// TIA Portal V20 export
FUNCTION "CollectAlarms" : Void   // FC71, LAD
TITLE = U1Em7_SepaPnp
// stored: Namespace Unit1.Em7, SetENOAutomatically false
   VAR_INPUT
      resetAlarms : Bool;
      disableAlarms : Bool;
   END_VAR
   VAR_OUTPUT
      commandsToUnit : "LUC_typeStateCommands";   // Feedback to the unit
   END_VAR
   VAR CONSTANT
      DelayTime : Time := T#300ms;
      NoDelayTime : Time;
   END_VAR
BEGIN

REGION Network 1: Reset Alarms
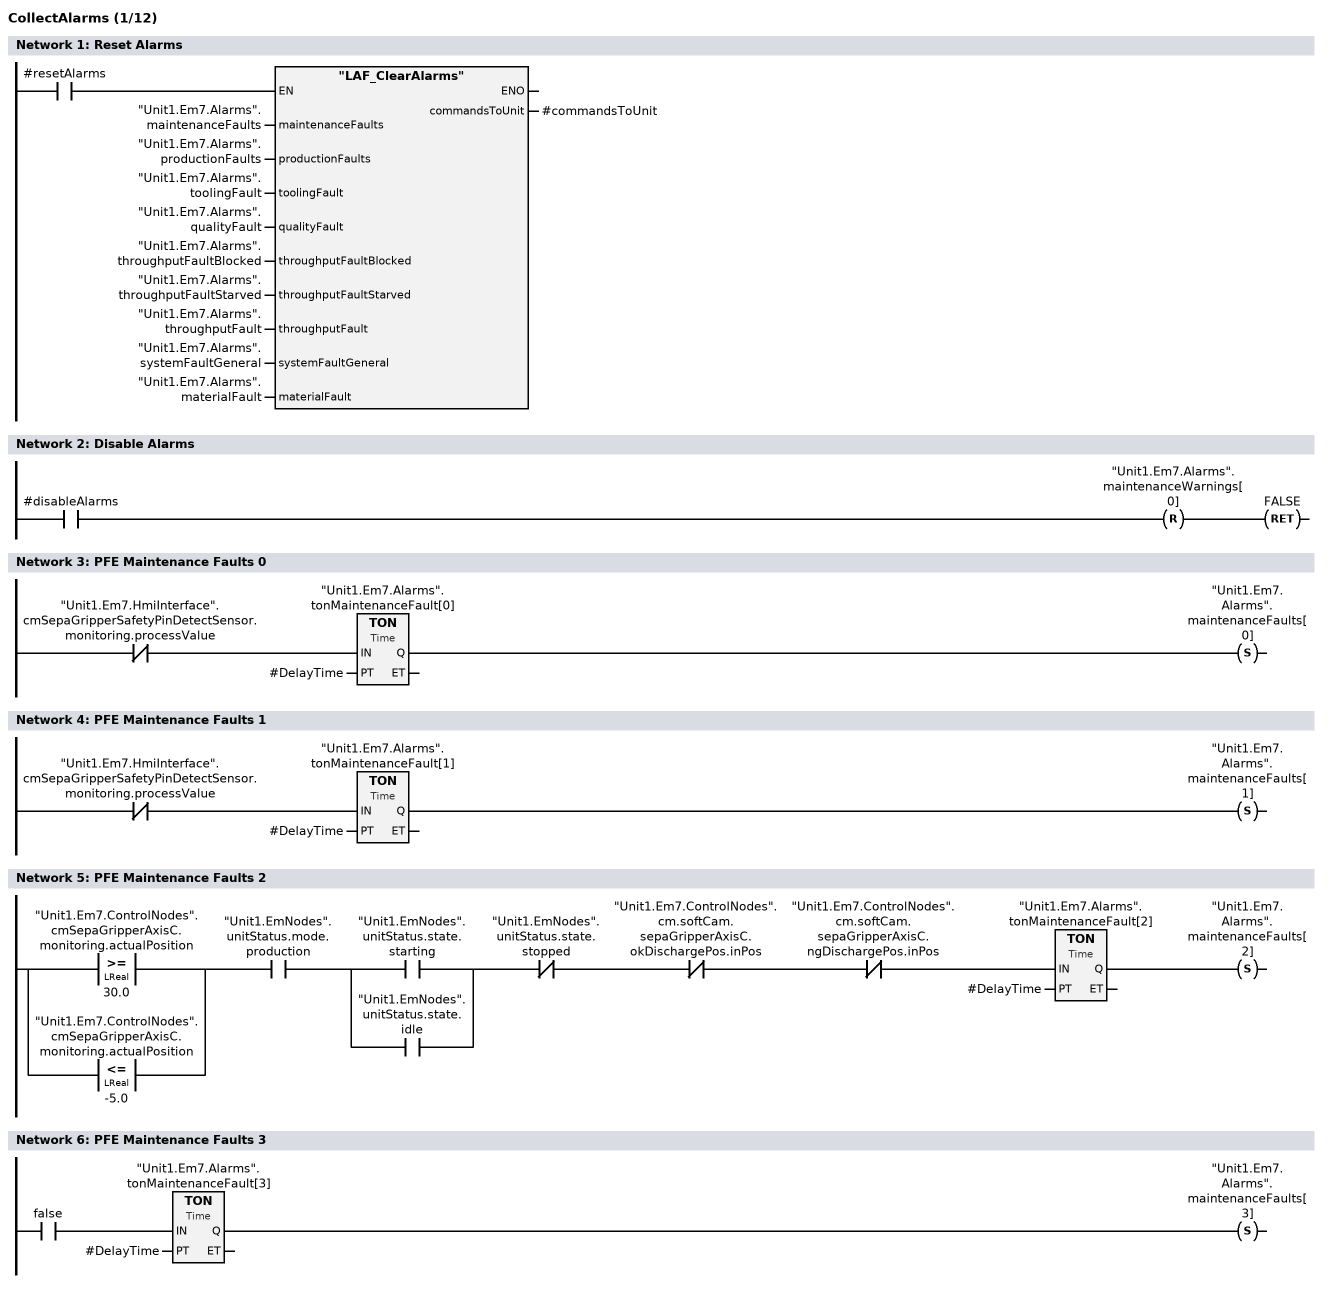
   RUNG wire#powerrail
      Contact( #resetAlarms )
      "LAF_ClearAlarms"(maintenanceFaults := "Unit1.Em7.Alarms".maintenanceFaults, productionFaults := "Unit1.Em7.Alarms".productionFaults, toolingFault := "Unit1.Em7.Alarms".toolingFault, qualityFault := "Unit1.Em7.Alarms".qualityFault, throughputFaultBlocked := "Unit1.Em7.Alarms".throughputFaultBlocked, throughputFaultStarved := "Unit1.Em7.Alarms".throughputFaultStarved, throughputFault := "Unit1.Em7.Alarms".throughputFault, systemFaultGeneral := "Unit1.Em7.Alarms".systemFaultGeneral, materialFault := "Unit1.Em7.Alarms".materialFault, commandsToUnit => #commandsToUnit)
   END_RUNG
   // the same network as SCL:
   IF #resetAlarms THEN
       "LAF_ClearAlarms"(maintenanceFaults := "Unit1.Em7.Alarms".maintenanceFaults,
                         productionFaults := "Unit1.Em7.Alarms".productionFaults,
                         toolingFault := "Unit1.Em7.Alarms".toolingFault,
                         qualityFault := "Unit1.Em7.Alarms".qualityFault,
                         throughputFaultBlocked := "Unit1.Em7.Alarms".throughputFaultBlocked,
                         throughputFaultStarved := "Unit1.Em7.Alarms".throughputFaultStarved,
                         throughputFault := "Unit1.Em7.Alarms".throughputFault,
                         systemFaultGeneral := "Unit1.Em7.Alarms".systemFaultGeneral,
                         materialFault := "Unit1.Em7.Alarms".materialFault,
                         commandsToUnit => #commandsToUnit);
   END_IF;
END_REGION

REGION Network 2: Disable Alarms
   RUNG wire#powerrail
      Contact( #disableAlarms )
      R_Coil( "Unit1.Em7.Alarms".maintenanceWarnings[0] )
      ReturnCoil( FALSE )
   END_RUNG
   // the same network as SCL:
   IF #disableAlarms THEN
       "Unit1.Em7.Alarms".maintenanceWarnings[0] := FALSE;
       ENO := FALSE;
       RETURN;
   END_IF;
END_REGION

REGION Network 3: PFE Maintenance Faults 0
   RUNG wire#powerrail
      I_Contact( "Unit1.Em7.HmiInterface".cmSepaGripperSafetyPinDetectSensor.monitoring.processValue )
      { S7_Templates := "time_type := Time" } "Unit1.Em7.Alarms".tonMaintenanceFault[0].TON(pt := #DelayTime, et =>)
      S_Coil( "Unit1.Em7.Alarms".maintenanceFaults[0] )
   END_RUNG
   // the same network as SCL:
   "Unit1.Em7.Alarms".tonMaintenanceFault[0].TON(IN := NOT "Unit1.Em7.HmiInterface".cmSepaGripperSafetyPinDetectSensor.monitoring.processValue,
                           PT := #DelayTime);
   IF "Unit1.Em7.Alarms".tonMaintenanceFault[0].Q THEN
       "Unit1.Em7.Alarms".maintenanceFaults[0] := TRUE;
   END_IF;
END_REGION

REGION Network 4: PFE Maintenance Faults 1
   RUNG wire#powerrail
      I_Contact( "Unit1.Em7.HmiInterface".cmSepaGripperSafetyPinDetectSensor.monitoring.processValue )
      { S7_Templates := "time_type := Time" } "Unit1.Em7.Alarms".tonMaintenanceFault[1].TON(pt := #DelayTime, et =>)
      S_Coil( "Unit1.Em7.Alarms".maintenanceFaults[1] )
   END_RUNG
   // the same network as SCL:
   "Unit1.Em7.Alarms".tonMaintenanceFault[1].TON(IN := NOT "Unit1.Em7.HmiInterface".cmSepaGripperSafetyPinDetectSensor.monitoring.processValue,
                           PT := #DelayTime);
   IF "Unit1.Em7.Alarms".tonMaintenanceFault[1].Q THEN
       "Unit1.Em7.Alarms".maintenanceFaults[1] := TRUE;
   END_IF;
END_REGION

REGION Network 5: PFE Maintenance Faults 2
   RUNG wire#powerrail
      { S7_Templates := "SrcType := LReal" } GE_Contact(in1 := "Unit1.Em7.ControlNodes".cmSepaGripperAxisC.monitoring.actualPosition, in2 := 30.0)
      wire#w1
      Contact( "Unit1.EmNodes".unitStatus.mode.production )
      wire#w2
      Contact( "Unit1.EmNodes".unitStatus.state.starting )
      wire#w3
      I_Contact( "Unit1.EmNodes".unitStatus.state.stopped )
      I_Contact( "Unit1.Em7.ControlNodes".cm.softCam.sepaGripperAxisC.okDischargePos.inPos )
      I_Contact( "Unit1.Em7.ControlNodes".cm.softCam.sepaGripperAxisC.ngDischargePos.inPos )
      { S7_Templates := "time_type := Time" } "Unit1.Em7.Alarms".tonMaintenanceFault[2].TON(pt := #DelayTime, et =>)
      S_Coil( "Unit1.Em7.Alarms".maintenanceFaults[2] )
   END_RUNG
   RUNG wire#powerrail
      { S7_Templates := "SrcType := LReal" } LE_Contact(in1 := "Unit1.Em7.ControlNodes".cmSepaGripperAxisC.monitoring.actualPosition, in2 := -5.0)
   END_RUNG wire#w1
   RUNG wire#w2
      Contact( "Unit1.EmNodes".unitStatus.state.idle )
   END_RUNG wire#w3
   // the same network as SCL:
   "Unit1.Em7.Alarms".tonMaintenanceFault[2].TON(IN := (("Unit1.Em7.ControlNodes".cmSepaGripperAxisC.monitoring.actualPosition >= 30.0) OR ("Unit1.Em7.ControlNodes".cmSepaGripperAxisC.monitoring.actualPosition <= (-5.0))) AND "Unit1.EmNodes".unitStatus.mode.production AND ("Unit1.EmNodes".unitStatus.state.starting OR "Unit1.EmNodes".unitStatus.state.idle) AND NOT "Unit1.EmNodes".unitStatus.state.stopped AND NOT "Unit1.Em7.ControlNodes".cm.softCam.sepaGripperAxisC.okDischargePos.inPos AND NOT "Unit1.Em7.ControlNodes".cm.softCam.sepaGripperAxisC.ngDischargePos.inPos,
                           PT := #DelayTime);
   IF "Unit1.Em7.Alarms".tonMaintenanceFault[2].Q THEN
       "Unit1.Em7.Alarms".maintenanceFaults[2] := TRUE;
   END_IF;
END_REGION

REGION Network 6: PFE Maintenance Faults 3
   RUNG wire#powerrail
      Contact( false )
      { S7_Templates := "time_type := Time" } "Unit1.Em7.Alarms".tonMaintenanceFault[3].TON(pt := #DelayTime, et =>)
      S_Coil( "Unit1.Em7.Alarms".maintenanceFaults[3] )
   END_RUNG
   // the same network as SCL:
   "Unit1.Em7.Alarms".tonMaintenanceFault[3].TON(IN := false, PT := #DelayTime);
   IF "Unit1.Em7.Alarms".tonMaintenanceFault[3].Q THEN
       "Unit1.Em7.Alarms".maintenanceFaults[3] := TRUE;
   END_IF;
END_REGION

REGION Network 7: PFE Maintenance Faults 4
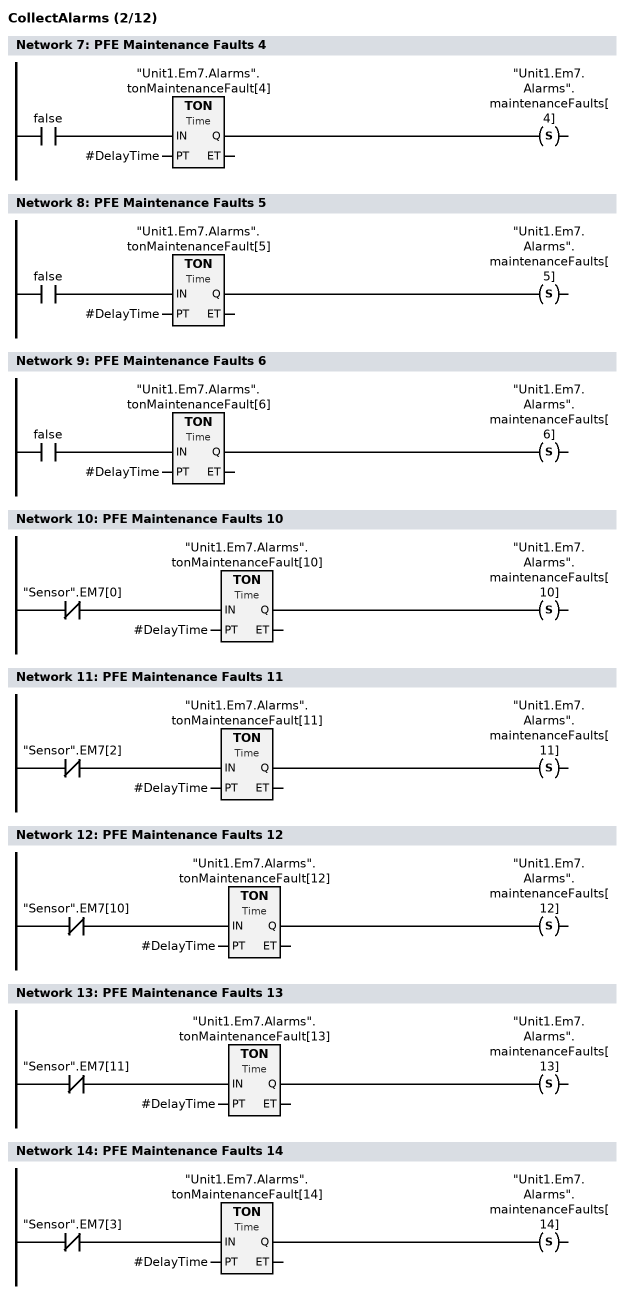
   RUNG wire#powerrail
      Contact( false )
      { S7_Templates := "time_type := Time" } "Unit1.Em7.Alarms".tonMaintenanceFault[4].TON(pt := #DelayTime, et =>)
      S_Coil( "Unit1.Em7.Alarms".maintenanceFaults[4] )
   END_RUNG
   // the same network as SCL:
   "Unit1.Em7.Alarms".tonMaintenanceFault[4].TON(IN := false, PT := #DelayTime);
   IF "Unit1.Em7.Alarms".tonMaintenanceFault[4].Q THEN
       "Unit1.Em7.Alarms".maintenanceFaults[4] := TRUE;
   END_IF;
END_REGION

REGION Network 8: PFE Maintenance Faults 5
   RUNG wire#powerrail
      Contact( false )
      { S7_Templates := "time_type := Time" } "Unit1.Em7.Alarms".tonMaintenanceFault[5].TON(pt := #DelayTime, et =>)
      S_Coil( "Unit1.Em7.Alarms".maintenanceFaults[5] )
   END_RUNG
   // the same network as SCL:
   "Unit1.Em7.Alarms".tonMaintenanceFault[5].TON(IN := false, PT := #DelayTime);
   IF "Unit1.Em7.Alarms".tonMaintenanceFault[5].Q THEN
       "Unit1.Em7.Alarms".maintenanceFaults[5] := TRUE;
   END_IF;
END_REGION

REGION Network 9: PFE Maintenance Faults 6
   RUNG wire#powerrail
      Contact( false )
      { S7_Templates := "time_type := Time" } "Unit1.Em7.Alarms".tonMaintenanceFault[6].TON(pt := #DelayTime, et =>)
      S_Coil( "Unit1.Em7.Alarms".maintenanceFaults[6] )
   END_RUNG
   // the same network as SCL:
   "Unit1.Em7.Alarms".tonMaintenanceFault[6].TON(IN := false, PT := #DelayTime);
   IF "Unit1.Em7.Alarms".tonMaintenanceFault[6].Q THEN
       "Unit1.Em7.Alarms".maintenanceFaults[6] := TRUE;
   END_IF;
END_REGION

REGION Network 10: PFE Maintenance Faults 10
   RUNG wire#powerrail
      I_Contact( "Sensor".EM7[0] )
      { S7_Templates := "time_type := Time" } "Unit1.Em7.Alarms".tonMaintenanceFault[10].TON(pt := #DelayTime, et =>)
      S_Coil( "Unit1.Em7.Alarms".maintenanceFaults[10] )
   END_RUNG
   // the same network as SCL:
   "Unit1.Em7.Alarms".tonMaintenanceFault[10].TON(IN := NOT "Sensor".EM7[0], PT := #DelayTime);
   IF "Unit1.Em7.Alarms".tonMaintenanceFault[10].Q THEN
       "Unit1.Em7.Alarms".maintenanceFaults[10] := TRUE;
   END_IF;
END_REGION

REGION Network 11: PFE Maintenance Faults 11
   RUNG wire#powerrail
      I_Contact( "Sensor".EM7[2] )
      { S7_Templates := "time_type := Time" } "Unit1.Em7.Alarms".tonMaintenanceFault[11].TON(pt := #DelayTime, et =>)
      S_Coil( "Unit1.Em7.Alarms".maintenanceFaults[11] )
   END_RUNG
   // the same network as SCL:
   "Unit1.Em7.Alarms".tonMaintenanceFault[11].TON(IN := NOT "Sensor".EM7[2], PT := #DelayTime);
   IF "Unit1.Em7.Alarms".tonMaintenanceFault[11].Q THEN
       "Unit1.Em7.Alarms".maintenanceFaults[11] := TRUE;
   END_IF;
END_REGION

REGION Network 12: PFE Maintenance Faults 12
   RUNG wire#powerrail
      I_Contact( "Sensor".EM7[10] )
      { S7_Templates := "time_type := Time" } "Unit1.Em7.Alarms".tonMaintenanceFault[12].TON(pt := #DelayTime, et =>)
      S_Coil( "Unit1.Em7.Alarms".maintenanceFaults[12] )
   END_RUNG
   // the same network as SCL:
   "Unit1.Em7.Alarms".tonMaintenanceFault[12].TON(IN := NOT "Sensor".EM7[10], PT := #DelayTime);
   IF "Unit1.Em7.Alarms".tonMaintenanceFault[12].Q THEN
       "Unit1.Em7.Alarms".maintenanceFaults[12] := TRUE;
   END_IF;
END_REGION

REGION Network 13: PFE Maintenance Faults 13
   RUNG wire#powerrail
      I_Contact( "Sensor".EM7[11] )
      { S7_Templates := "time_type := Time" } "Unit1.Em7.Alarms".tonMaintenanceFault[13].TON(pt := #DelayTime, et =>)
      S_Coil( "Unit1.Em7.Alarms".maintenanceFaults[13] )
   END_RUNG
   // the same network as SCL:
   "Unit1.Em7.Alarms".tonMaintenanceFault[13].TON(IN := NOT "Sensor".EM7[11], PT := #DelayTime);
   IF "Unit1.Em7.Alarms".tonMaintenanceFault[13].Q THEN
       "Unit1.Em7.Alarms".maintenanceFaults[13] := TRUE;
   END_IF;
END_REGION

REGION Network 14: PFE Maintenance Faults 14
   RUNG wire#powerrail
      I_Contact( "Sensor".EM7[3] )
      { S7_Templates := "time_type := Time" } "Unit1.Em7.Alarms".tonMaintenanceFault[14].TON(pt := #DelayTime, et =>)
      S_Coil( "Unit1.Em7.Alarms".maintenanceFaults[14] )
   END_RUNG
   // the same network as SCL:
   "Unit1.Em7.Alarms".tonMaintenanceFault[14].TON(IN := NOT "Sensor".EM7[3], PT := #DelayTime);
   IF "Unit1.Em7.Alarms".tonMaintenanceFault[14].Q THEN
       "Unit1.Em7.Alarms".maintenanceFaults[14] := TRUE;
   END_IF;
END_REGION

REGION Network 15: PFE Maintenance Faults 15
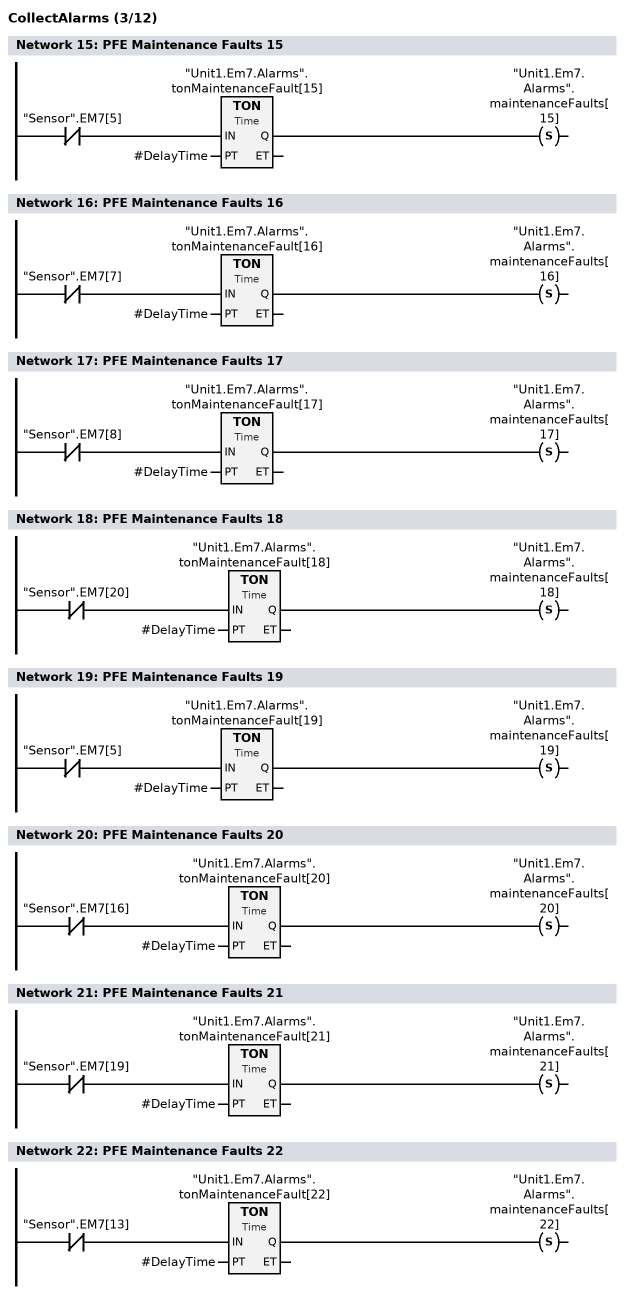
   RUNG wire#powerrail
      I_Contact( "Sensor".EM7[5] )
      { S7_Templates := "time_type := Time" } "Unit1.Em7.Alarms".tonMaintenanceFault[15].TON(pt := #DelayTime, et =>)
      S_Coil( "Unit1.Em7.Alarms".maintenanceFaults[15] )
   END_RUNG
   // the same network as SCL:
   "Unit1.Em7.Alarms".tonMaintenanceFault[15].TON(IN := NOT "Sensor".EM7[5], PT := #DelayTime);
   IF "Unit1.Em7.Alarms".tonMaintenanceFault[15].Q THEN
       "Unit1.Em7.Alarms".maintenanceFaults[15] := TRUE;
   END_IF;
END_REGION

REGION Network 16: PFE Maintenance Faults 16
   RUNG wire#powerrail
      I_Contact( "Sensor".EM7[7] )
      { S7_Templates := "time_type := Time" } "Unit1.Em7.Alarms".tonMaintenanceFault[16].TON(pt := #DelayTime, et =>)
      S_Coil( "Unit1.Em7.Alarms".maintenanceFaults[16] )
   END_RUNG
   // the same network as SCL:
   "Unit1.Em7.Alarms".tonMaintenanceFault[16].TON(IN := NOT "Sensor".EM7[7], PT := #DelayTime);
   IF "Unit1.Em7.Alarms".tonMaintenanceFault[16].Q THEN
       "Unit1.Em7.Alarms".maintenanceFaults[16] := TRUE;
   END_IF;
END_REGION

REGION Network 17: PFE Maintenance Faults 17
   RUNG wire#powerrail
      I_Contact( "Sensor".EM7[8] )
      { S7_Templates := "time_type := Time" } "Unit1.Em7.Alarms".tonMaintenanceFault[17].TON(pt := #DelayTime, et =>)
      S_Coil( "Unit1.Em7.Alarms".maintenanceFaults[17] )
   END_RUNG
   // the same network as SCL:
   "Unit1.Em7.Alarms".tonMaintenanceFault[17].TON(IN := NOT "Sensor".EM7[8], PT := #DelayTime);
   IF "Unit1.Em7.Alarms".tonMaintenanceFault[17].Q THEN
       "Unit1.Em7.Alarms".maintenanceFaults[17] := TRUE;
   END_IF;
END_REGION

REGION Network 18: PFE Maintenance Faults 18
   RUNG wire#powerrail
      I_Contact( "Sensor".EM7[20] )
      { S7_Templates := "time_type := Time" } "Unit1.Em7.Alarms".tonMaintenanceFault[18].TON(pt := #DelayTime, et =>)
      S_Coil( "Unit1.Em7.Alarms".maintenanceFaults[18] )
   END_RUNG
   // the same network as SCL:
   "Unit1.Em7.Alarms".tonMaintenanceFault[18].TON(IN := NOT "Sensor".EM7[20], PT := #DelayTime);
   IF "Unit1.Em7.Alarms".tonMaintenanceFault[18].Q THEN
       "Unit1.Em7.Alarms".maintenanceFaults[18] := TRUE;
   END_IF;
END_REGION

REGION Network 19: PFE Maintenance Faults 19
   RUNG wire#powerrail
      I_Contact( "Sensor".EM7[5] )
      { S7_Templates := "time_type := Time" } "Unit1.Em7.Alarms".tonMaintenanceFault[19].TON(pt := #DelayTime, et =>)
      S_Coil( "Unit1.Em7.Alarms".maintenanceFaults[19] )
   END_RUNG
   // the same network as SCL:
   "Unit1.Em7.Alarms".tonMaintenanceFault[19].TON(IN := NOT "Sensor".EM7[5], PT := #DelayTime);
   IF "Unit1.Em7.Alarms".tonMaintenanceFault[19].Q THEN
       "Unit1.Em7.Alarms".maintenanceFaults[19] := TRUE;
   END_IF;
END_REGION

REGION Network 20: PFE Maintenance Faults 20
   RUNG wire#powerrail
      I_Contact( "Sensor".EM7[16] )
      { S7_Templates := "time_type := Time" } "Unit1.Em7.Alarms".tonMaintenanceFault[20].TON(pt := #DelayTime, et =>)
      S_Coil( "Unit1.Em7.Alarms".maintenanceFaults[20] )
   END_RUNG
   // the same network as SCL:
   "Unit1.Em7.Alarms".tonMaintenanceFault[20].TON(IN := NOT "Sensor".EM7[16], PT := #DelayTime);
   IF "Unit1.Em7.Alarms".tonMaintenanceFault[20].Q THEN
       "Unit1.Em7.Alarms".maintenanceFaults[20] := TRUE;
   END_IF;
END_REGION

REGION Network 21: PFE Maintenance Faults 21
   RUNG wire#powerrail
      I_Contact( "Sensor".EM7[19] )
      { S7_Templates := "time_type := Time" } "Unit1.Em7.Alarms".tonMaintenanceFault[21].TON(pt := #DelayTime, et =>)
      S_Coil( "Unit1.Em7.Alarms".maintenanceFaults[21] )
   END_RUNG
   // the same network as SCL:
   "Unit1.Em7.Alarms".tonMaintenanceFault[21].TON(IN := NOT "Sensor".EM7[19], PT := #DelayTime);
   IF "Unit1.Em7.Alarms".tonMaintenanceFault[21].Q THEN
       "Unit1.Em7.Alarms".maintenanceFaults[21] := TRUE;
   END_IF;
END_REGION

REGION Network 22: PFE Maintenance Faults 22
   RUNG wire#powerrail
      I_Contact( "Sensor".EM7[13] )
      { S7_Templates := "time_type := Time" } "Unit1.Em7.Alarms".tonMaintenanceFault[22].TON(pt := #DelayTime, et =>)
      S_Coil( "Unit1.Em7.Alarms".maintenanceFaults[22] )
   END_RUNG
   // the same network as SCL:
   "Unit1.Em7.Alarms".tonMaintenanceFault[22].TON(IN := NOT "Sensor".EM7[13], PT := #DelayTime);
   IF "Unit1.Em7.Alarms".tonMaintenanceFault[22].Q THEN
       "Unit1.Em7.Alarms".maintenanceFaults[22] := TRUE;
   END_IF;
END_REGION

REGION Network 23: PFE Maintenance Faults 23
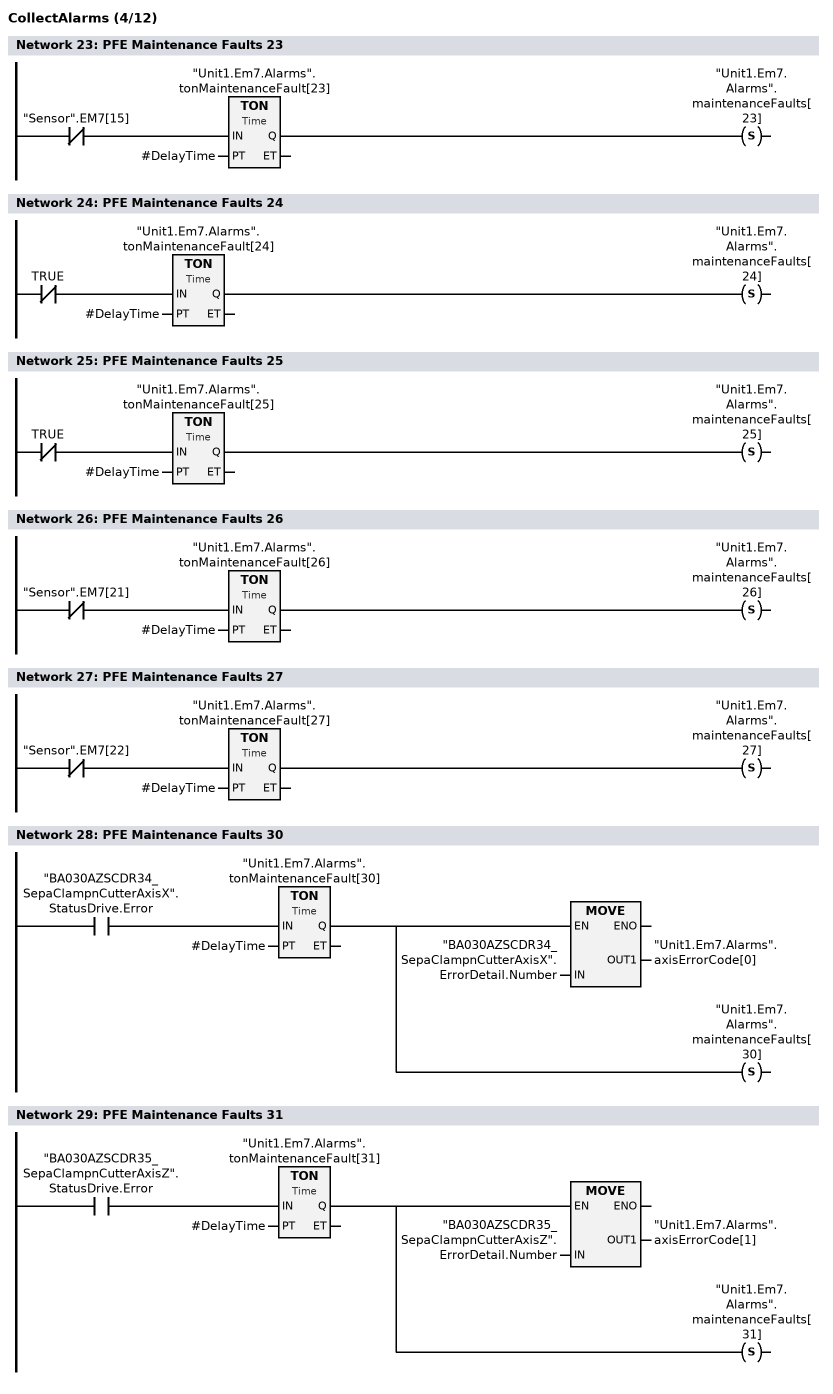
   RUNG wire#powerrail
      I_Contact( "Sensor".EM7[15] )
      { S7_Templates := "time_type := Time" } "Unit1.Em7.Alarms".tonMaintenanceFault[23].TON(pt := #DelayTime, et =>)
      S_Coil( "Unit1.Em7.Alarms".maintenanceFaults[23] )
   END_RUNG
   // the same network as SCL:
   "Unit1.Em7.Alarms".tonMaintenanceFault[23].TON(IN := NOT "Sensor".EM7[15], PT := #DelayTime);
   IF "Unit1.Em7.Alarms".tonMaintenanceFault[23].Q THEN
       "Unit1.Em7.Alarms".maintenanceFaults[23] := TRUE;
   END_IF;
END_REGION

REGION Network 24: PFE Maintenance Faults 24
   RUNG wire#powerrail
      I_Contact( TRUE )
      { S7_Templates := "time_type := Time" } "Unit1.Em7.Alarms".tonMaintenanceFault[24].TON(pt := #DelayTime, et =>)
      S_Coil( "Unit1.Em7.Alarms".maintenanceFaults[24] )
   END_RUNG
   // the same network as SCL:
   "Unit1.Em7.Alarms".tonMaintenanceFault[24].TON(IN := NOT TRUE, PT := #DelayTime);
   IF "Unit1.Em7.Alarms".tonMaintenanceFault[24].Q THEN
       "Unit1.Em7.Alarms".maintenanceFaults[24] := TRUE;
   END_IF;
END_REGION

REGION Network 25: PFE Maintenance Faults 25
   RUNG wire#powerrail
      I_Contact( TRUE )
      { S7_Templates := "time_type := Time" } "Unit1.Em7.Alarms".tonMaintenanceFault[25].TON(pt := #DelayTime, et =>)
      S_Coil( "Unit1.Em7.Alarms".maintenanceFaults[25] )
   END_RUNG
   // the same network as SCL:
   "Unit1.Em7.Alarms".tonMaintenanceFault[25].TON(IN := NOT TRUE, PT := #DelayTime);
   IF "Unit1.Em7.Alarms".tonMaintenanceFault[25].Q THEN
       "Unit1.Em7.Alarms".maintenanceFaults[25] := TRUE;
   END_IF;
END_REGION

REGION Network 26: PFE Maintenance Faults 26
   RUNG wire#powerrail
      I_Contact( "Sensor".EM7[21] )
      { S7_Templates := "time_type := Time" } "Unit1.Em7.Alarms".tonMaintenanceFault[26].TON(pt := #DelayTime, et =>)
      S_Coil( "Unit1.Em7.Alarms".maintenanceFaults[26] )
   END_RUNG
   // the same network as SCL:
   "Unit1.Em7.Alarms".tonMaintenanceFault[26].TON(IN := NOT "Sensor".EM7[21], PT := #DelayTime);
   IF "Unit1.Em7.Alarms".tonMaintenanceFault[26].Q THEN
       "Unit1.Em7.Alarms".maintenanceFaults[26] := TRUE;
   END_IF;
END_REGION

REGION Network 27: PFE Maintenance Faults 27
   RUNG wire#powerrail
      I_Contact( "Sensor".EM7[22] )
      { S7_Templates := "time_type := Time" } "Unit1.Em7.Alarms".tonMaintenanceFault[27].TON(pt := #DelayTime, et =>)
      S_Coil( "Unit1.Em7.Alarms".maintenanceFaults[27] )
   END_RUNG
   // the same network as SCL:
   "Unit1.Em7.Alarms".tonMaintenanceFault[27].TON(IN := NOT "Sensor".EM7[22], PT := #DelayTime);
   IF "Unit1.Em7.Alarms".tonMaintenanceFault[27].Q THEN
       "Unit1.Em7.Alarms".maintenanceFaults[27] := TRUE;
   END_IF;
END_REGION

REGION Network 28: PFE Maintenance Faults 30
   RUNG wire#powerrail
      Contact( "BA030AZSCDR34_SepaClampnCutterAxisX".StatusDrive.Error )
      { S7_Templates := "time_type := Time" } "Unit1.Em7.Alarms".tonMaintenanceFault[30].TON(pt := #DelayTime, et =>)
      wire#w1
      Move(in := "BA030AZSCDR34_SepaClampnCutterAxisX".ErrorDetail.Number, out1 => "Unit1.Em7.Alarms".axisErrorCode[0])
   END_RUNG
   RUNG wire#w1
      S_Coil( "Unit1.Em7.Alarms".maintenanceFaults[30] )
   END_RUNG
   // the same network as SCL:
   "Unit1.Em7.Alarms".tonMaintenanceFault[30].TON(IN := "BA030AZSCDR34_SepaClampnCutterAxisX".StatusDrive.Error,
                           PT := #DelayTime);
   IF "Unit1.Em7.Alarms".tonMaintenanceFault[30].Q THEN
       "Unit1.Em7.Alarms".axisErrorCode[0] := "BA030AZSCDR34_SepaClampnCutterAxisX".ErrorDetail.Number;
       "Unit1.Em7.Alarms".maintenanceFaults[30] := TRUE;
   END_IF;
END_REGION

REGION Network 29: PFE Maintenance Faults 31
   RUNG wire#powerrail
      Contact( "BA030AZSCDR35_SepaClampnCutterAxisZ".StatusDrive.Error )
      { S7_Templates := "time_type := Time" } "Unit1.Em7.Alarms".tonMaintenanceFault[31].TON(pt := #DelayTime, et =>)
      wire#w1
      Move(in := "BA030AZSCDR35_SepaClampnCutterAxisZ".ErrorDetail.Number, out1 => "Unit1.Em7.Alarms".axisErrorCode[1])
   END_RUNG
   RUNG wire#w1
      S_Coil( "Unit1.Em7.Alarms".maintenanceFaults[31] )
   END_RUNG
   // the same network as SCL:
   "Unit1.Em7.Alarms".tonMaintenanceFault[31].TON(IN := "BA030AZSCDR35_SepaClampnCutterAxisZ".StatusDrive.Error,
                           PT := #DelayTime);
   IF "Unit1.Em7.Alarms".tonMaintenanceFault[31].Q THEN
       "Unit1.Em7.Alarms".axisErrorCode[1] := "BA030AZSCDR35_SepaClampnCutterAxisZ".ErrorDetail.Number;
       "Unit1.Em7.Alarms".maintenanceFaults[31] := TRUE;
   END_IF;
END_REGION

REGION Network 30: PFE Maintenance Faults 32
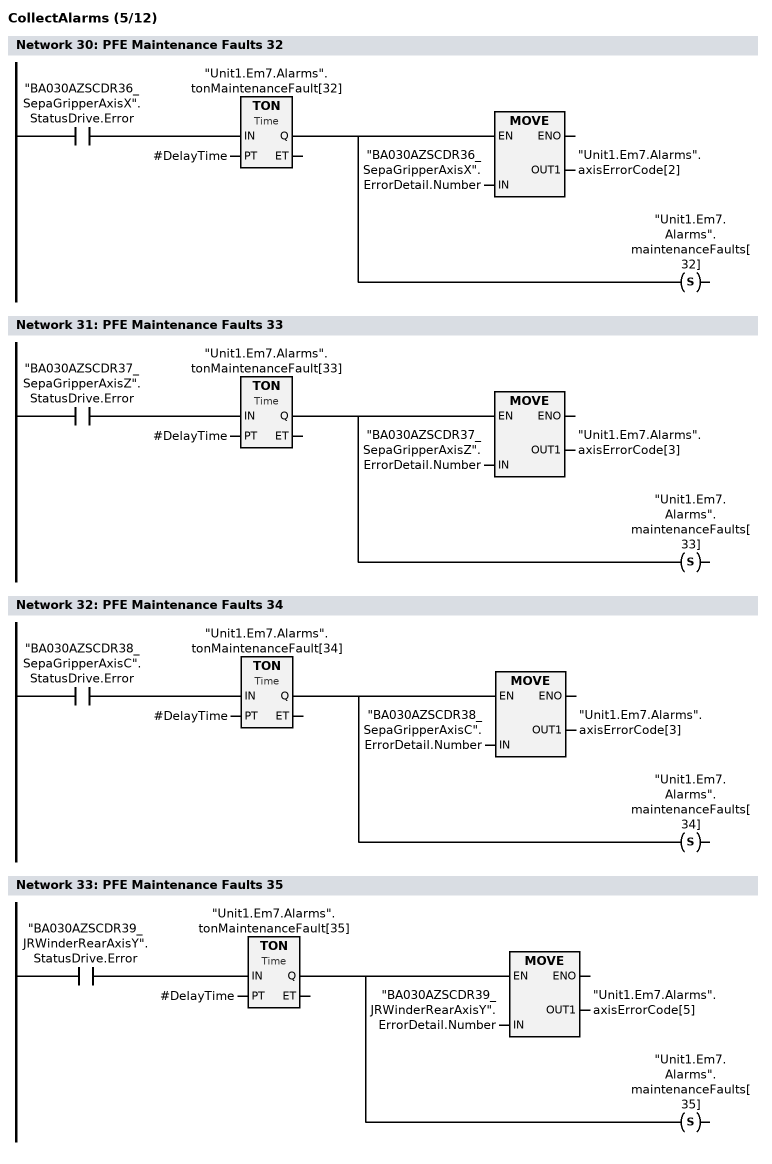
   RUNG wire#powerrail
      Contact( "BA030AZSCDR36_SepaGripperAxisX".StatusDrive.Error )
      { S7_Templates := "time_type := Time" } "Unit1.Em7.Alarms".tonMaintenanceFault[32].TON(pt := #DelayTime, et =>)
      wire#w1
      Move(in := "BA030AZSCDR36_SepaGripperAxisX".ErrorDetail.Number, out1 => "Unit1.Em7.Alarms".axisErrorCode[2])
   END_RUNG
   RUNG wire#w1
      S_Coil( "Unit1.Em7.Alarms".maintenanceFaults[32] )
   END_RUNG
   // the same network as SCL:
   "Unit1.Em7.Alarms".tonMaintenanceFault[32].TON(IN := "BA030AZSCDR36_SepaGripperAxisX".StatusDrive.Error,
                           PT := #DelayTime);
   IF "Unit1.Em7.Alarms".tonMaintenanceFault[32].Q THEN
       "Unit1.Em7.Alarms".axisErrorCode[2] := "BA030AZSCDR36_SepaGripperAxisX".ErrorDetail.Number;
       "Unit1.Em7.Alarms".maintenanceFaults[32] := TRUE;
   END_IF;
END_REGION

REGION Network 31: PFE Maintenance Faults 33
   RUNG wire#powerrail
      Contact( "BA030AZSCDR37_SepaGripperAxisZ".StatusDrive.Error )
      { S7_Templates := "time_type := Time" } "Unit1.Em7.Alarms".tonMaintenanceFault[33].TON(pt := #DelayTime, et =>)
      wire#w1
      Move(in := "BA030AZSCDR37_SepaGripperAxisZ".ErrorDetail.Number, out1 => "Unit1.Em7.Alarms".axisErrorCode[3])
   END_RUNG
   RUNG wire#w1
      S_Coil( "Unit1.Em7.Alarms".maintenanceFaults[33] )
   END_RUNG
   // the same network as SCL:
   "Unit1.Em7.Alarms".tonMaintenanceFault[33].TON(IN := "BA030AZSCDR37_SepaGripperAxisZ".StatusDrive.Error,
                           PT := #DelayTime);
   IF "Unit1.Em7.Alarms".tonMaintenanceFault[33].Q THEN
       "Unit1.Em7.Alarms".axisErrorCode[3] := "BA030AZSCDR37_SepaGripperAxisZ".ErrorDetail.Number;
       "Unit1.Em7.Alarms".maintenanceFaults[33] := TRUE;
   END_IF;
END_REGION

REGION Network 32: PFE Maintenance Faults 34
   RUNG wire#powerrail
      Contact( "BA030AZSCDR38_SepaGripperAxisC".StatusDrive.Error )
      { S7_Templates := "time_type := Time" } "Unit1.Em7.Alarms".tonMaintenanceFault[34].TON(pt := #DelayTime, et =>)
      wire#w1
      Move(in := "BA030AZSCDR38_SepaGripperAxisC".ErrorDetail.Number, out1 => "Unit1.Em7.Alarms".axisErrorCode[3])
   END_RUNG
   RUNG wire#w1
      S_Coil( "Unit1.Em7.Alarms".maintenanceFaults[34] )
   END_RUNG
   // the same network as SCL:
   "Unit1.Em7.Alarms".tonMaintenanceFault[34].TON(IN := "BA030AZSCDR38_SepaGripperAxisC".StatusDrive.Error,
                           PT := #DelayTime);
   IF "Unit1.Em7.Alarms".tonMaintenanceFault[34].Q THEN
       "Unit1.Em7.Alarms".axisErrorCode[3] := "BA030AZSCDR38_SepaGripperAxisC".ErrorDetail.Number;
       "Unit1.Em7.Alarms".maintenanceFaults[34] := TRUE;
   END_IF;
END_REGION

REGION Network 33: PFE Maintenance Faults 35
   RUNG wire#powerrail
      Contact( "BA030AZSCDR39_JRWinderRearAxisY".StatusDrive.Error )
      { S7_Templates := "time_type := Time" } "Unit1.Em7.Alarms".tonMaintenanceFault[35].TON(pt := #DelayTime, et =>)
      wire#w1
      Move(in := "BA030AZSCDR39_JRWinderRearAxisY".ErrorDetail.Number, out1 => "Unit1.Em7.Alarms".axisErrorCode[5])
   END_RUNG
   RUNG wire#w1
      S_Coil( "Unit1.Em7.Alarms".maintenanceFaults[35] )
   END_RUNG
   // the same network as SCL:
   "Unit1.Em7.Alarms".tonMaintenanceFault[35].TON(IN := "BA030AZSCDR39_JRWinderRearAxisY".StatusDrive.Error,
                           PT := #DelayTime);
   IF "Unit1.Em7.Alarms".tonMaintenanceFault[35].Q THEN
       "Unit1.Em7.Alarms".axisErrorCode[5] := "BA030AZSCDR39_JRWinderRearAxisY".ErrorDetail.Number;
       "Unit1.Em7.Alarms".maintenanceFaults[35] := TRUE;
   END_IF;
END_REGION

REGION Network 34: PFE Maintenance Faults 36
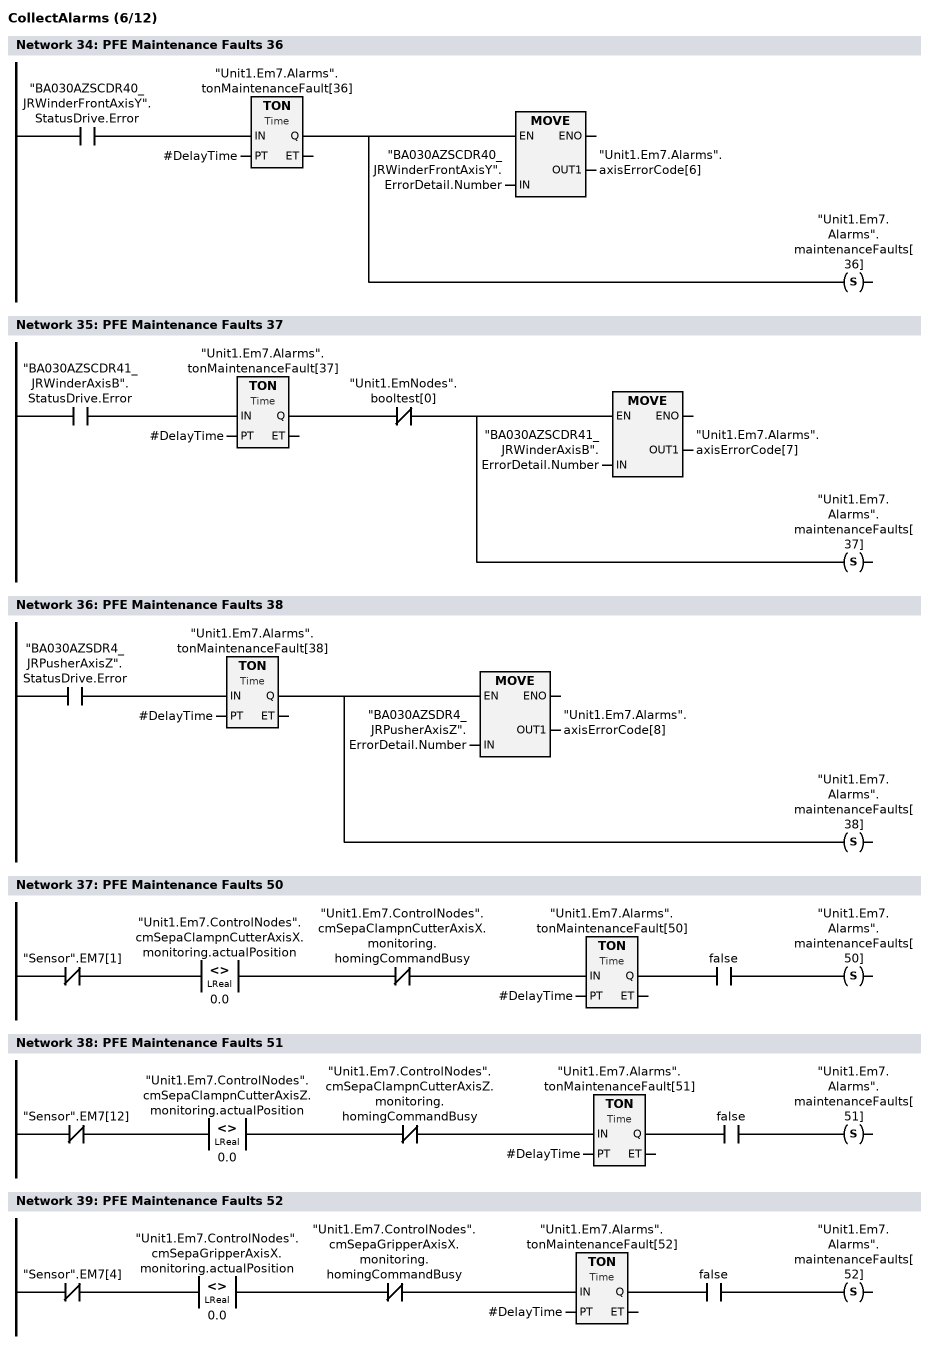
   RUNG wire#powerrail
      Contact( "BA030AZSCDR40_JRWinderFrontAxisY".StatusDrive.Error )
      { S7_Templates := "time_type := Time" } "Unit1.Em7.Alarms".tonMaintenanceFault[36].TON(pt := #DelayTime, et =>)
      wire#w1
      Move(in := "BA030AZSCDR40_JRWinderFrontAxisY".ErrorDetail.Number, out1 => "Unit1.Em7.Alarms".axisErrorCode[6])
   END_RUNG
   RUNG wire#w1
      S_Coil( "Unit1.Em7.Alarms".maintenanceFaults[36] )
   END_RUNG
   // the same network as SCL:
   "Unit1.Em7.Alarms".tonMaintenanceFault[36].TON(IN := "BA030AZSCDR40_JRWinderFrontAxisY".StatusDrive.Error,
                           PT := #DelayTime);
   IF "Unit1.Em7.Alarms".tonMaintenanceFault[36].Q THEN
       "Unit1.Em7.Alarms".axisErrorCode[6] := "BA030AZSCDR40_JRWinderFrontAxisY".ErrorDetail.Number;
       "Unit1.Em7.Alarms".maintenanceFaults[36] := TRUE;
   END_IF;
END_REGION

REGION Network 35: PFE Maintenance Faults 37
   RUNG wire#powerrail
      Contact( "BA030AZSCDR41_JRWinderAxisB".StatusDrive.Error )
      { S7_Templates := "time_type := Time" } "Unit1.Em7.Alarms".tonMaintenanceFault[37].TON(pt := #DelayTime, et =>)
      I_Contact( "Unit1.EmNodes".booltest[0] )
      wire#w1
      Move(in := "BA030AZSCDR41_JRWinderAxisB".ErrorDetail.Number, out1 => "Unit1.Em7.Alarms".axisErrorCode[7])
   END_RUNG
   RUNG wire#w1
      S_Coil( "Unit1.Em7.Alarms".maintenanceFaults[37] )
   END_RUNG
   // the same network as SCL:
   "Unit1.Em7.Alarms".tonMaintenanceFault[37].TON(IN := "BA030AZSCDR41_JRWinderAxisB".StatusDrive.Error,
                           PT := #DelayTime);
   IF "Unit1.Em7.Alarms".tonMaintenanceFault[37].Q AND NOT "Unit1.EmNodes".booltest[0] THEN
       "Unit1.Em7.Alarms".axisErrorCode[7] := "BA030AZSCDR41_JRWinderAxisB".ErrorDetail.Number;
       "Unit1.Em7.Alarms".maintenanceFaults[37] := TRUE;
   END_IF;
END_REGION

REGION Network 36: PFE Maintenance Faults 38
   RUNG wire#powerrail
      Contact( "BA030AZSDR4_JRPusherAxisZ".StatusDrive.Error )
      { S7_Templates := "time_type := Time" } "Unit1.Em7.Alarms".tonMaintenanceFault[38].TON(pt := #DelayTime, et =>)
      wire#w1
      Move(in := "BA030AZSDR4_JRPusherAxisZ".ErrorDetail.Number, out1 => "Unit1.Em7.Alarms".axisErrorCode[8])
   END_RUNG
   RUNG wire#w1
      S_Coil( "Unit1.Em7.Alarms".maintenanceFaults[38] )
   END_RUNG
   // the same network as SCL:
   "Unit1.Em7.Alarms".tonMaintenanceFault[38].TON(IN := "BA030AZSDR4_JRPusherAxisZ".StatusDrive.Error,
                           PT := #DelayTime);
   IF "Unit1.Em7.Alarms".tonMaintenanceFault[38].Q THEN
       "Unit1.Em7.Alarms".axisErrorCode[8] := "BA030AZSDR4_JRPusherAxisZ".ErrorDetail.Number;
       "Unit1.Em7.Alarms".maintenanceFaults[38] := TRUE;
   END_IF;
END_REGION

REGION Network 37: PFE Maintenance Faults 50
   RUNG wire#powerrail
      I_Contact( "Sensor".EM7[1] )
      { S7_Templates := "SrcType := LReal" } NE_Contact(in1 := "Unit1.Em7.ControlNodes".cmSepaClampnCutterAxisX.monitoring.actualPosition, in2 := 0.0)
      I_Contact( "Unit1.Em7.ControlNodes".cmSepaClampnCutterAxisX.monitoring.homingCommandBusy )
      { S7_Templates := "time_type := Time" } "Unit1.Em7.Alarms".tonMaintenanceFault[50].TON(pt := #DelayTime, et =>)
      Contact( false )
      S_Coil( "Unit1.Em7.Alarms".maintenanceFaults[50] )
   END_RUNG
   // the same network as SCL:
   "Unit1.Em7.Alarms".tonMaintenanceFault[50].TON(IN := NOT "Sensor".EM7[1] AND ("Unit1.Em7.ControlNodes".cmSepaClampnCutterAxisX.monitoring.actualPosition <> 0.0) AND NOT "Unit1.Em7.ControlNodes".cmSepaClampnCutterAxisX.monitoring.homingCommandBusy,
                           PT := #DelayTime);
   IF "Unit1.Em7.Alarms".tonMaintenanceFault[50].Q AND false THEN
       "Unit1.Em7.Alarms".maintenanceFaults[50] := TRUE;
   END_IF;
END_REGION

REGION Network 38: PFE Maintenance Faults 51
   RUNG wire#powerrail
      I_Contact( "Sensor".EM7[12] )
      { S7_Templates := "SrcType := LReal" } NE_Contact(in1 := "Unit1.Em7.ControlNodes".cmSepaClampnCutterAxisZ.monitoring.actualPosition, in2 := 0.0)
      I_Contact( "Unit1.Em7.ControlNodes".cmSepaClampnCutterAxisZ.monitoring.homingCommandBusy )
      { S7_Templates := "time_type := Time" } "Unit1.Em7.Alarms".tonMaintenanceFault[51].TON(pt := #DelayTime, et =>)
      Contact( false )
      S_Coil( "Unit1.Em7.Alarms".maintenanceFaults[51] )
   END_RUNG
   // the same network as SCL:
   "Unit1.Em7.Alarms".tonMaintenanceFault[51].TON(IN := NOT "Sensor".EM7[12] AND ("Unit1.Em7.ControlNodes".cmSepaClampnCutterAxisZ.monitoring.actualPosition <> 0.0) AND NOT "Unit1.Em7.ControlNodes".cmSepaClampnCutterAxisZ.monitoring.homingCommandBusy,
                           PT := #DelayTime);
   IF "Unit1.Em7.Alarms".tonMaintenanceFault[51].Q AND false THEN
       "Unit1.Em7.Alarms".maintenanceFaults[51] := TRUE;
   END_IF;
END_REGION

REGION Network 39: PFE Maintenance Faults 52
   RUNG wire#powerrail
      I_Contact( "Sensor".EM7[4] )
      { S7_Templates := "SrcType := LReal" } NE_Contact(in1 := "Unit1.Em7.ControlNodes".cmSepaGripperAxisX.monitoring.actualPosition, in2 := 0.0)
      I_Contact( "Unit1.Em7.ControlNodes".cmSepaGripperAxisX.monitoring.homingCommandBusy )
      { S7_Templates := "time_type := Time" } "Unit1.Em7.Alarms".tonMaintenanceFault[52].TON(pt := #DelayTime, et =>)
      Contact( false )
      S_Coil( "Unit1.Em7.Alarms".maintenanceFaults[52] )
   END_RUNG
   // the same network as SCL:
   "Unit1.Em7.Alarms".tonMaintenanceFault[52].TON(IN := NOT "Sensor".EM7[4] AND ("Unit1.Em7.ControlNodes".cmSepaGripperAxisX.monitoring.actualPosition <> 0.0) AND NOT "Unit1.Em7.ControlNodes".cmSepaGripperAxisX.monitoring.homingCommandBusy,
                           PT := #DelayTime);
   IF "Unit1.Em7.Alarms".tonMaintenanceFault[52].Q AND false THEN
       "Unit1.Em7.Alarms".maintenanceFaults[52] := TRUE;
   END_IF;
END_REGION

REGION Network 40: PFE Maintenance Faults 53
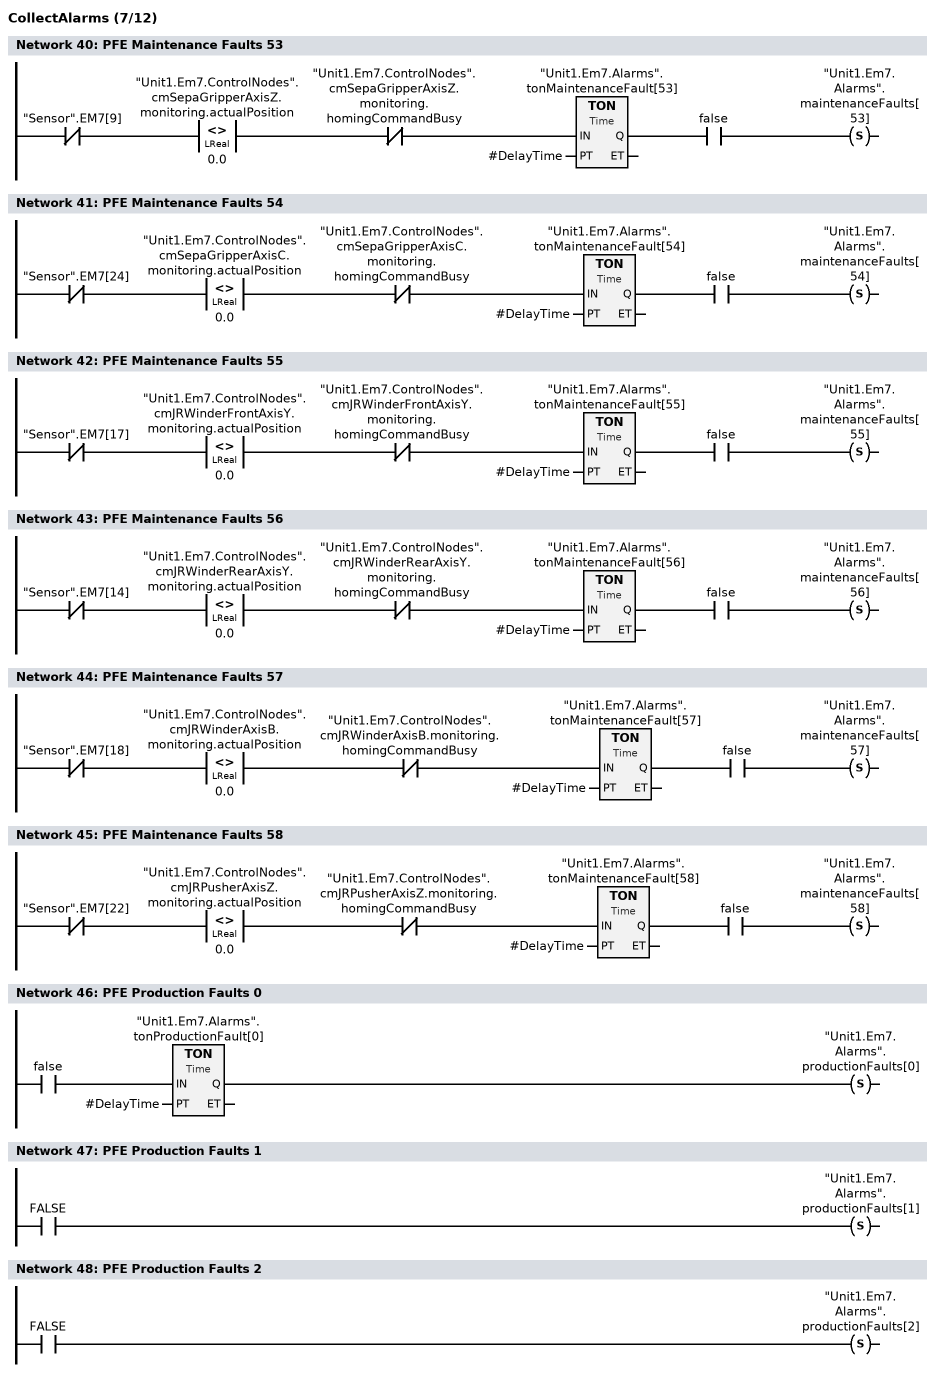
   RUNG wire#powerrail
      I_Contact( "Sensor".EM7[9] )
      { S7_Templates := "SrcType := LReal" } NE_Contact(in1 := "Unit1.Em7.ControlNodes".cmSepaGripperAxisZ.monitoring.actualPosition, in2 := 0.0)
      I_Contact( "Unit1.Em7.ControlNodes".cmSepaGripperAxisZ.monitoring.homingCommandBusy )
      { S7_Templates := "time_type := Time" } "Unit1.Em7.Alarms".tonMaintenanceFault[53].TON(pt := #DelayTime, et =>)
      Contact( false )
      S_Coil( "Unit1.Em7.Alarms".maintenanceFaults[53] )
   END_RUNG
   // the same network as SCL:
   "Unit1.Em7.Alarms".tonMaintenanceFault[53].TON(IN := NOT "Sensor".EM7[9] AND ("Unit1.Em7.ControlNodes".cmSepaGripperAxisZ.monitoring.actualPosition <> 0.0) AND NOT "Unit1.Em7.ControlNodes".cmSepaGripperAxisZ.monitoring.homingCommandBusy,
                           PT := #DelayTime);
   IF "Unit1.Em7.Alarms".tonMaintenanceFault[53].Q AND false THEN
       "Unit1.Em7.Alarms".maintenanceFaults[53] := TRUE;
   END_IF;
END_REGION

REGION Network 41: PFE Maintenance Faults 54
   RUNG wire#powerrail
      I_Contact( "Sensor".EM7[24] )
      { S7_Templates := "SrcType := LReal" } NE_Contact(in1 := "Unit1.Em7.ControlNodes".cmSepaGripperAxisC.monitoring.actualPosition, in2 := 0.0)
      I_Contact( "Unit1.Em7.ControlNodes".cmSepaGripperAxisC.monitoring.homingCommandBusy )
      { S7_Templates := "time_type := Time" } "Unit1.Em7.Alarms".tonMaintenanceFault[54].TON(pt := #DelayTime, et =>)
      Contact( false )
      S_Coil( "Unit1.Em7.Alarms".maintenanceFaults[54] )
   END_RUNG
   // the same network as SCL:
   "Unit1.Em7.Alarms".tonMaintenanceFault[54].TON(IN := NOT "Sensor".EM7[24] AND ("Unit1.Em7.ControlNodes".cmSepaGripperAxisC.monitoring.actualPosition <> 0.0) AND NOT "Unit1.Em7.ControlNodes".cmSepaGripperAxisC.monitoring.homingCommandBusy,
                           PT := #DelayTime);
   IF "Unit1.Em7.Alarms".tonMaintenanceFault[54].Q AND false THEN
       "Unit1.Em7.Alarms".maintenanceFaults[54] := TRUE;
   END_IF;
END_REGION

REGION Network 42: PFE Maintenance Faults 55
   RUNG wire#powerrail
      I_Contact( "Sensor".EM7[17] )
      { S7_Templates := "SrcType := LReal" } NE_Contact(in1 := "Unit1.Em7.ControlNodes".cmJRWinderFrontAxisY.monitoring.actualPosition, in2 := 0.0)
      I_Contact( "Unit1.Em7.ControlNodes".cmJRWinderFrontAxisY.monitoring.homingCommandBusy )
      { S7_Templates := "time_type := Time" } "Unit1.Em7.Alarms".tonMaintenanceFault[55].TON(pt := #DelayTime, et =>)
      Contact( false )
      S_Coil( "Unit1.Em7.Alarms".maintenanceFaults[55] )
   END_RUNG
   // the same network as SCL:
   "Unit1.Em7.Alarms".tonMaintenanceFault[55].TON(IN := NOT "Sensor".EM7[17] AND ("Unit1.Em7.ControlNodes".cmJRWinderFrontAxisY.monitoring.actualPosition <> 0.0) AND NOT "Unit1.Em7.ControlNodes".cmJRWinderFrontAxisY.monitoring.homingCommandBusy,
                           PT := #DelayTime);
   IF "Unit1.Em7.Alarms".tonMaintenanceFault[55].Q AND false THEN
       "Unit1.Em7.Alarms".maintenanceFaults[55] := TRUE;
   END_IF;
END_REGION

REGION Network 43: PFE Maintenance Faults 56
   RUNG wire#powerrail
      I_Contact( "Sensor".EM7[14] )
      { S7_Templates := "SrcType := LReal" } NE_Contact(in1 := "Unit1.Em7.ControlNodes".cmJRWinderRearAxisY.monitoring.actualPosition, in2 := 0.0)
      I_Contact( "Unit1.Em7.ControlNodes".cmJRWinderRearAxisY.monitoring.homingCommandBusy )
      { S7_Templates := "time_type := Time" } "Unit1.Em7.Alarms".tonMaintenanceFault[56].TON(pt := #DelayTime, et =>)
      Contact( false )
      S_Coil( "Unit1.Em7.Alarms".maintenanceFaults[56] )
   END_RUNG
   // the same network as SCL:
   "Unit1.Em7.Alarms".tonMaintenanceFault[56].TON(IN := NOT "Sensor".EM7[14] AND ("Unit1.Em7.ControlNodes".cmJRWinderRearAxisY.monitoring.actualPosition <> 0.0) AND NOT "Unit1.Em7.ControlNodes".cmJRWinderRearAxisY.monitoring.homingCommandBusy,
                           PT := #DelayTime);
   IF "Unit1.Em7.Alarms".tonMaintenanceFault[56].Q AND false THEN
       "Unit1.Em7.Alarms".maintenanceFaults[56] := TRUE;
   END_IF;
END_REGION

REGION Network 44: PFE Maintenance Faults 57
   RUNG wire#powerrail
      I_Contact( "Sensor".EM7[18] )
      { S7_Templates := "SrcType := LReal" } NE_Contact(in1 := "Unit1.Em7.ControlNodes".cmJRWinderAxisB.monitoring.actualPosition, in2 := 0.0)
      I_Contact( "Unit1.Em7.ControlNodes".cmJRWinderAxisB.monitoring.homingCommandBusy )
      { S7_Templates := "time_type := Time" } "Unit1.Em7.Alarms".tonMaintenanceFault[57].TON(pt := #DelayTime, et =>)
      Contact( false )
      S_Coil( "Unit1.Em7.Alarms".maintenanceFaults[57] )
   END_RUNG
   // the same network as SCL:
   "Unit1.Em7.Alarms".tonMaintenanceFault[57].TON(IN := NOT "Sensor".EM7[18] AND ("Unit1.Em7.ControlNodes".cmJRWinderAxisB.monitoring.actualPosition <> 0.0) AND NOT "Unit1.Em7.ControlNodes".cmJRWinderAxisB.monitoring.homingCommandBusy,
                           PT := #DelayTime);
   IF "Unit1.Em7.Alarms".tonMaintenanceFault[57].Q AND false THEN
       "Unit1.Em7.Alarms".maintenanceFaults[57] := TRUE;
   END_IF;
END_REGION

REGION Network 45: PFE Maintenance Faults 58
   RUNG wire#powerrail
      I_Contact( "Sensor".EM7[22] )
      { S7_Templates := "SrcType := LReal" } NE_Contact(in1 := "Unit1.Em7.ControlNodes".cmJRPusherAxisZ.monitoring.actualPosition, in2 := 0.0)
      I_Contact( "Unit1.Em7.ControlNodes".cmJRPusherAxisZ.monitoring.homingCommandBusy )
      { S7_Templates := "time_type := Time" } "Unit1.Em7.Alarms".tonMaintenanceFault[58].TON(pt := #DelayTime, et =>)
      Contact( false )
      S_Coil( "Unit1.Em7.Alarms".maintenanceFaults[58] )
   END_RUNG
   // the same network as SCL:
   "Unit1.Em7.Alarms".tonMaintenanceFault[58].TON(IN := NOT "Sensor".EM7[22] AND ("Unit1.Em7.ControlNodes".cmJRPusherAxisZ.monitoring.actualPosition <> 0.0) AND NOT "Unit1.Em7.ControlNodes".cmJRPusherAxisZ.monitoring.homingCommandBusy,
                           PT := #DelayTime);
   IF "Unit1.Em7.Alarms".tonMaintenanceFault[58].Q AND false THEN
       "Unit1.Em7.Alarms".maintenanceFaults[58] := TRUE;
   END_IF;
END_REGION

REGION Network 46: PFE Production Faults 0
   RUNG wire#powerrail
      Contact( false )
      { S7_Templates := "time_type := Time" } "Unit1.Em7.Alarms".tonProductionFault[0].TON(pt := #DelayTime, et =>)
      S_Coil( "Unit1.Em7.Alarms".productionFaults[0] )
   END_RUNG
   // the same network as SCL:
   "Unit1.Em7.Alarms".tonProductionFault[0].TON(IN := false, PT := #DelayTime);
   IF "Unit1.Em7.Alarms".tonProductionFault[0].Q THEN "Unit1.Em7.Alarms".productionFaults[0] := TRUE; END_IF;
END_REGION

REGION Network 47: PFE Production Faults 1
   RUNG wire#powerrail
      Contact( FALSE )
      S_Coil( "Unit1.Em7.Alarms".productionFaults[1] )
   END_RUNG
   // the same network as SCL:
   IF FALSE THEN "Unit1.Em7.Alarms".productionFaults[1] := TRUE; END_IF;
END_REGION

REGION Network 48: PFE Production Faults 2
   RUNG wire#powerrail
      Contact( FALSE )
      S_Coil( "Unit1.Em7.Alarms".productionFaults[2] )
   END_RUNG
   // the same network as SCL:
   IF FALSE THEN "Unit1.Em7.Alarms".productionFaults[2] := TRUE; END_IF;
END_REGION

REGION Network 49: PFE Production Faults 3
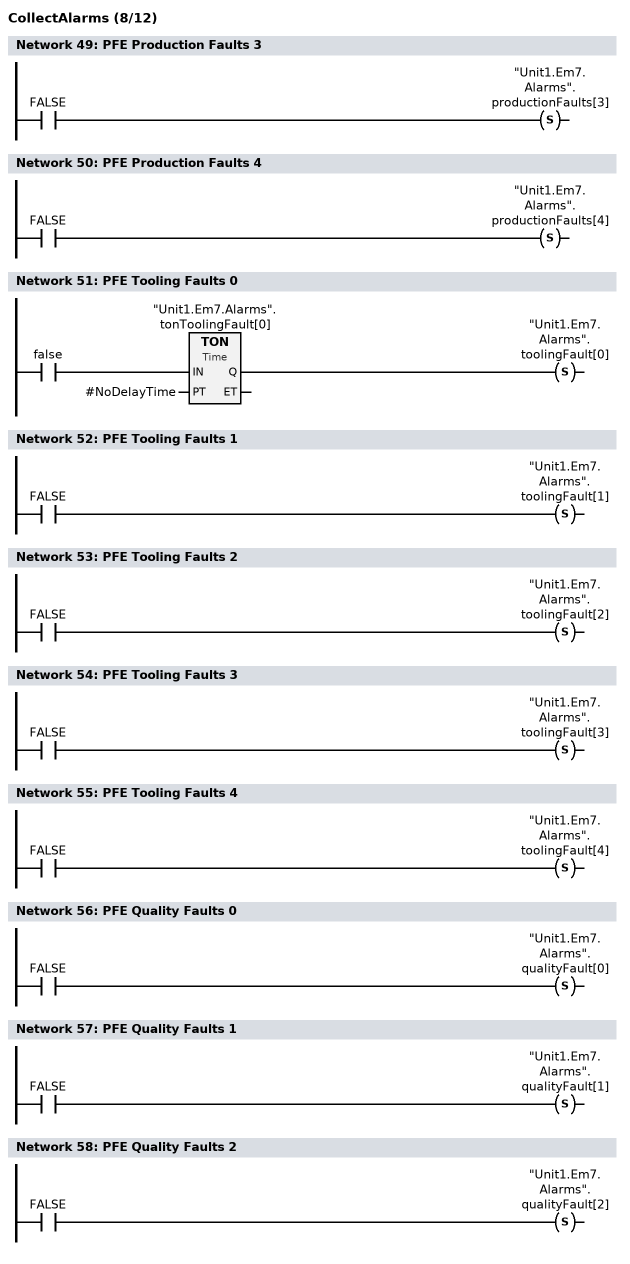
   RUNG wire#powerrail
      Contact( FALSE )
      S_Coil( "Unit1.Em7.Alarms".productionFaults[3] )
   END_RUNG
   // the same network as SCL:
   IF FALSE THEN "Unit1.Em7.Alarms".productionFaults[3] := TRUE; END_IF;
END_REGION

REGION Network 50: PFE Production Faults 4
   RUNG wire#powerrail
      Contact( FALSE )
      S_Coil( "Unit1.Em7.Alarms".productionFaults[4] )
   END_RUNG
   // the same network as SCL:
   IF FALSE THEN "Unit1.Em7.Alarms".productionFaults[4] := TRUE; END_IF;
END_REGION

REGION Network 51: PFE Tooling Faults 0
   RUNG wire#powerrail
      Contact( false )
      { S7_Templates := "time_type := Time" } "Unit1.Em7.Alarms".tonToolingFault[0].TON(pt := #NoDelayTime, et =>)
      S_Coil( "Unit1.Em7.Alarms".toolingFault[0] )
   END_RUNG
   // the same network as SCL:
   "Unit1.Em7.Alarms".tonToolingFault[0].TON(IN := false, PT := #NoDelayTime);
   IF "Unit1.Em7.Alarms".tonToolingFault[0].Q THEN "Unit1.Em7.Alarms".toolingFault[0] := TRUE; END_IF;
END_REGION

REGION Network 52: PFE Tooling Faults 1
   RUNG wire#powerrail
      Contact( FALSE )
      S_Coil( "Unit1.Em7.Alarms".toolingFault[1] )
   END_RUNG
   // the same network as SCL:
   IF FALSE THEN "Unit1.Em7.Alarms".toolingFault[1] := TRUE; END_IF;
END_REGION

REGION Network 53: PFE Tooling Faults 2
   RUNG wire#powerrail
      Contact( FALSE )
      S_Coil( "Unit1.Em7.Alarms".toolingFault[2] )
   END_RUNG
   // the same network as SCL:
   IF FALSE THEN "Unit1.Em7.Alarms".toolingFault[2] := TRUE; END_IF;
END_REGION

REGION Network 54: PFE Tooling Faults 3
   RUNG wire#powerrail
      Contact( FALSE )
      S_Coil( "Unit1.Em7.Alarms".toolingFault[3] )
   END_RUNG
   // the same network as SCL:
   IF FALSE THEN "Unit1.Em7.Alarms".toolingFault[3] := TRUE; END_IF;
END_REGION

REGION Network 55: PFE Tooling Faults 4
   RUNG wire#powerrail
      Contact( FALSE )
      S_Coil( "Unit1.Em7.Alarms".toolingFault[4] )
   END_RUNG
   // the same network as SCL:
   IF FALSE THEN "Unit1.Em7.Alarms".toolingFault[4] := TRUE; END_IF;
END_REGION

REGION Network 56: PFE Quality Faults 0
   RUNG wire#powerrail
      Contact( FALSE )
      S_Coil( "Unit1.Em7.Alarms".qualityFault[0] )
   END_RUNG
   // the same network as SCL:
   IF FALSE THEN "Unit1.Em7.Alarms".qualityFault[0] := TRUE; END_IF;
END_REGION

REGION Network 57: PFE Quality Faults 1
   RUNG wire#powerrail
      Contact( FALSE )
      S_Coil( "Unit1.Em7.Alarms".qualityFault[1] )
   END_RUNG
   // the same network as SCL:
   IF FALSE THEN "Unit1.Em7.Alarms".qualityFault[1] := TRUE; END_IF;
END_REGION

REGION Network 58: PFE Quality Faults 2
   RUNG wire#powerrail
      Contact( FALSE )
      S_Coil( "Unit1.Em7.Alarms".qualityFault[2] )
   END_RUNG
   // the same network as SCL:
   IF FALSE THEN "Unit1.Em7.Alarms".qualityFault[2] := TRUE; END_IF;
END_REGION

REGION Network 59: PFE Quality Faults 3
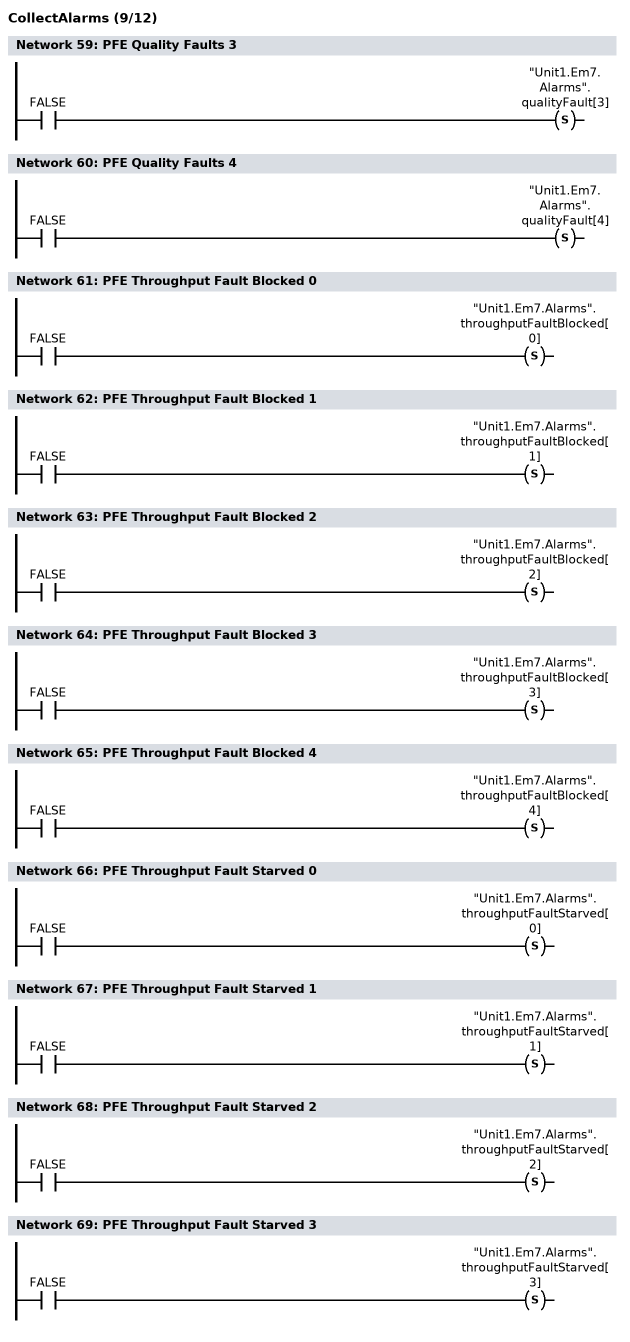
   RUNG wire#powerrail
      Contact( FALSE )
      S_Coil( "Unit1.Em7.Alarms".qualityFault[3] )
   END_RUNG
   // the same network as SCL:
   IF FALSE THEN "Unit1.Em7.Alarms".qualityFault[3] := TRUE; END_IF;
END_REGION

REGION Network 60: PFE Quality Faults 4
   RUNG wire#powerrail
      Contact( FALSE )
      S_Coil( "Unit1.Em7.Alarms".qualityFault[4] )
   END_RUNG
   // the same network as SCL:
   IF FALSE THEN "Unit1.Em7.Alarms".qualityFault[4] := TRUE; END_IF;
END_REGION

REGION Network 61: PFE Throughput Fault Blocked 0
   RUNG wire#powerrail
      Contact( FALSE )
      S_Coil( "Unit1.Em7.Alarms".throughputFaultBlocked[0] )
   END_RUNG
   // the same network as SCL:
   IF FALSE THEN "Unit1.Em7.Alarms".throughputFaultBlocked[0] := TRUE; END_IF;
END_REGION

REGION Network 62: PFE Throughput Fault Blocked 1
   RUNG wire#powerrail
      Contact( FALSE )
      S_Coil( "Unit1.Em7.Alarms".throughputFaultBlocked[1] )
   END_RUNG
   // the same network as SCL:
   IF FALSE THEN "Unit1.Em7.Alarms".throughputFaultBlocked[1] := TRUE; END_IF;
END_REGION

REGION Network 63: PFE Throughput Fault Blocked 2
   RUNG wire#powerrail
      Contact( FALSE )
      S_Coil( "Unit1.Em7.Alarms".throughputFaultBlocked[2] )
   END_RUNG
   // the same network as SCL:
   IF FALSE THEN "Unit1.Em7.Alarms".throughputFaultBlocked[2] := TRUE; END_IF;
END_REGION

REGION Network 64: PFE Throughput Fault Blocked 3
   RUNG wire#powerrail
      Contact( FALSE )
      S_Coil( "Unit1.Em7.Alarms".throughputFaultBlocked[3] )
   END_RUNG
   // the same network as SCL:
   IF FALSE THEN "Unit1.Em7.Alarms".throughputFaultBlocked[3] := TRUE; END_IF;
END_REGION

REGION Network 65: PFE Throughput Fault Blocked 4
   RUNG wire#powerrail
      Contact( FALSE )
      S_Coil( "Unit1.Em7.Alarms".throughputFaultBlocked[4] )
   END_RUNG
   // the same network as SCL:
   IF FALSE THEN "Unit1.Em7.Alarms".throughputFaultBlocked[4] := TRUE; END_IF;
END_REGION

REGION Network 66: PFE Throughput Fault Starved 0
   RUNG wire#powerrail
      Contact( FALSE )
      S_Coil( "Unit1.Em7.Alarms".throughputFaultStarved[0] )
   END_RUNG
   // the same network as SCL:
   IF FALSE THEN "Unit1.Em7.Alarms".throughputFaultStarved[0] := TRUE; END_IF;
END_REGION

REGION Network 67: PFE Throughput Fault Starved 1
   RUNG wire#powerrail
      Contact( FALSE )
      S_Coil( "Unit1.Em7.Alarms".throughputFaultStarved[1] )
   END_RUNG
   // the same network as SCL:
   IF FALSE THEN "Unit1.Em7.Alarms".throughputFaultStarved[1] := TRUE; END_IF;
END_REGION

REGION Network 68: PFE Throughput Fault Starved 2
   RUNG wire#powerrail
      Contact( FALSE )
      S_Coil( "Unit1.Em7.Alarms".throughputFaultStarved[2] )
   END_RUNG
   // the same network as SCL:
   IF FALSE THEN "Unit1.Em7.Alarms".throughputFaultStarved[2] := TRUE; END_IF;
END_REGION

REGION Network 69: PFE Throughput Fault Starved 3
   RUNG wire#powerrail
      Contact( FALSE )
      S_Coil( "Unit1.Em7.Alarms".throughputFaultStarved[3] )
   END_RUNG
   // the same network as SCL:
   IF FALSE THEN "Unit1.Em7.Alarms".throughputFaultStarved[3] := TRUE; END_IF;
END_REGION

REGION Network 70: PFE Throughput Fault Starved 4
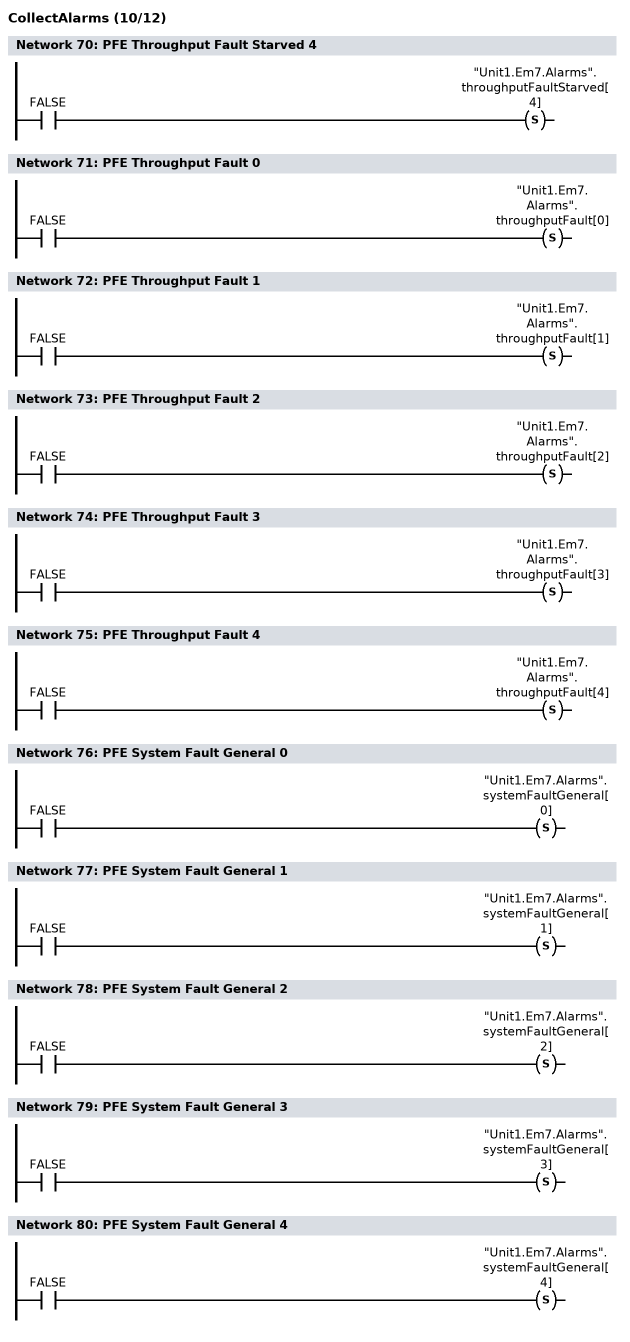
   RUNG wire#powerrail
      Contact( FALSE )
      S_Coil( "Unit1.Em7.Alarms".throughputFaultStarved[4] )
   END_RUNG
   // the same network as SCL:
   IF FALSE THEN "Unit1.Em7.Alarms".throughputFaultStarved[4] := TRUE; END_IF;
END_REGION

REGION Network 71: PFE Throughput Fault 0
   RUNG wire#powerrail
      Contact( FALSE )
      S_Coil( "Unit1.Em7.Alarms".throughputFault[0] )
   END_RUNG
   // the same network as SCL:
   IF FALSE THEN "Unit1.Em7.Alarms".throughputFault[0] := TRUE; END_IF;
END_REGION

REGION Network 72: PFE Throughput Fault 1
   RUNG wire#powerrail
      Contact( FALSE )
      S_Coil( "Unit1.Em7.Alarms".throughputFault[1] )
   END_RUNG
   // the same network as SCL:
   IF FALSE THEN "Unit1.Em7.Alarms".throughputFault[1] := TRUE; END_IF;
END_REGION

REGION Network 73: PFE Throughput Fault 2
   RUNG wire#powerrail
      Contact( FALSE )
      S_Coil( "Unit1.Em7.Alarms".throughputFault[2] )
   END_RUNG
   // the same network as SCL:
   IF FALSE THEN "Unit1.Em7.Alarms".throughputFault[2] := TRUE; END_IF;
END_REGION

REGION Network 74: PFE Throughput Fault 3
   RUNG wire#powerrail
      Contact( FALSE )
      S_Coil( "Unit1.Em7.Alarms".throughputFault[3] )
   END_RUNG
   // the same network as SCL:
   IF FALSE THEN "Unit1.Em7.Alarms".throughputFault[3] := TRUE; END_IF;
END_REGION

REGION Network 75: PFE Throughput Fault 4
   RUNG wire#powerrail
      Contact( FALSE )
      S_Coil( "Unit1.Em7.Alarms".throughputFault[4] )
   END_RUNG
   // the same network as SCL:
   IF FALSE THEN "Unit1.Em7.Alarms".throughputFault[4] := TRUE; END_IF;
END_REGION

REGION Network 76: PFE System Fault General 0
   RUNG wire#powerrail
      Contact( FALSE )
      S_Coil( "Unit1.Em7.Alarms".systemFaultGeneral[0] )
   END_RUNG
   // the same network as SCL:
   IF FALSE THEN "Unit1.Em7.Alarms".systemFaultGeneral[0] := TRUE; END_IF;
END_REGION

REGION Network 77: PFE System Fault General 1
   RUNG wire#powerrail
      Contact( FALSE )
      S_Coil( "Unit1.Em7.Alarms".systemFaultGeneral[1] )
   END_RUNG
   // the same network as SCL:
   IF FALSE THEN "Unit1.Em7.Alarms".systemFaultGeneral[1] := TRUE; END_IF;
END_REGION

REGION Network 78: PFE System Fault General 2
   RUNG wire#powerrail
      Contact( FALSE )
      S_Coil( "Unit1.Em7.Alarms".systemFaultGeneral[2] )
   END_RUNG
   // the same network as SCL:
   IF FALSE THEN "Unit1.Em7.Alarms".systemFaultGeneral[2] := TRUE; END_IF;
END_REGION

REGION Network 79: PFE System Fault General 3
   RUNG wire#powerrail
      Contact( FALSE )
      S_Coil( "Unit1.Em7.Alarms".systemFaultGeneral[3] )
   END_RUNG
   // the same network as SCL:
   IF FALSE THEN "Unit1.Em7.Alarms".systemFaultGeneral[3] := TRUE; END_IF;
END_REGION

REGION Network 80: PFE System Fault General 4
   RUNG wire#powerrail
      Contact( FALSE )
      S_Coil( "Unit1.Em7.Alarms".systemFaultGeneral[4] )
   END_RUNG
   // the same network as SCL:
   IF FALSE THEN "Unit1.Em7.Alarms".systemFaultGeneral[4] := TRUE; END_IF;
END_REGION

REGION Network 81: PFE Material Fault 0
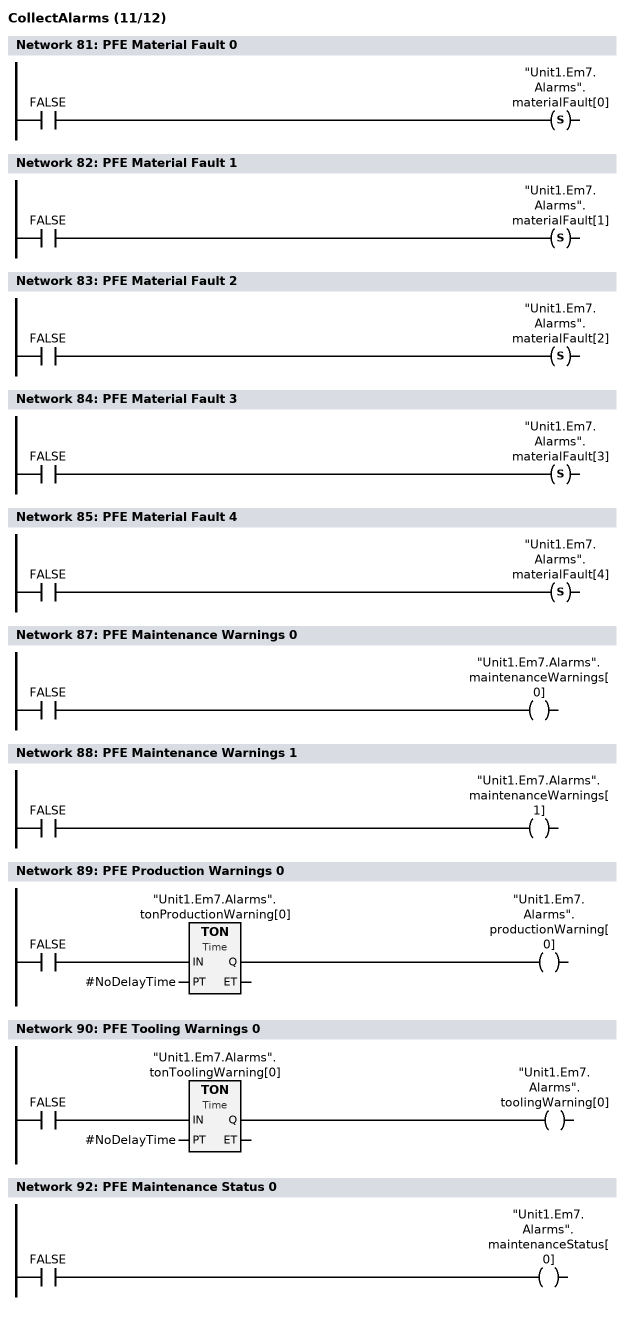
   RUNG wire#powerrail
      Contact( FALSE )
      S_Coil( "Unit1.Em7.Alarms".materialFault[0] )
   END_RUNG
   // the same network as SCL:
   IF FALSE THEN "Unit1.Em7.Alarms".materialFault[0] := TRUE; END_IF;
END_REGION

REGION Network 82: PFE Material Fault 1
   RUNG wire#powerrail
      Contact( FALSE )
      S_Coil( "Unit1.Em7.Alarms".materialFault[1] )
   END_RUNG
   // the same network as SCL:
   IF FALSE THEN "Unit1.Em7.Alarms".materialFault[1] := TRUE; END_IF;
END_REGION

REGION Network 83: PFE Material Fault 2
   RUNG wire#powerrail
      Contact( FALSE )
      S_Coil( "Unit1.Em7.Alarms".materialFault[2] )
   END_RUNG
   // the same network as SCL:
   IF FALSE THEN "Unit1.Em7.Alarms".materialFault[2] := TRUE; END_IF;
END_REGION

REGION Network 84: PFE Material Fault 3
   RUNG wire#powerrail
      Contact( FALSE )
      S_Coil( "Unit1.Em7.Alarms".materialFault[3] )
   END_RUNG
   // the same network as SCL:
   IF FALSE THEN "Unit1.Em7.Alarms".materialFault[3] := TRUE; END_IF;
END_REGION

REGION Network 85: PFE Material Fault 4
   RUNG wire#powerrail
      Contact( FALSE )
      S_Coil( "Unit1.Em7.Alarms".materialFault[4] )
   END_RUNG
   // the same network as SCL:
   IF FALSE THEN "Unit1.Em7.Alarms".materialFault[4] := TRUE; END_IF;
END_REGION

REGION Network 86: *************** Warning **************************
END_REGION

REGION Network 87: PFE Maintenance Warnings 0
   RUNG wire#powerrail
      Contact( FALSE )
      Coil( "Unit1.Em7.Alarms".maintenanceWarnings[0] )
   END_RUNG
   // the same network as SCL:
   "Unit1.Em7.Alarms".maintenanceWarnings[0] := FALSE;
END_REGION

REGION Network 88: PFE Maintenance Warnings 1
   RUNG wire#powerrail
      Contact( FALSE )
      Coil( "Unit1.Em7.Alarms".maintenanceWarnings[1] )
   END_RUNG
   // the same network as SCL:
   "Unit1.Em7.Alarms".maintenanceWarnings[1] := FALSE;
END_REGION

REGION Network 89: PFE Production Warnings 0
   RUNG wire#powerrail
      Contact( FALSE )
      { S7_Templates := "time_type := Time" } "Unit1.Em7.Alarms".tonProductionWarning[0].TON(pt := #NoDelayTime, et =>)
      Coil( "Unit1.Em7.Alarms".productionWarning[0] )
   END_RUNG
   // the same network as SCL:
   "Unit1.Em7.Alarms".tonProductionWarning[0].TON(IN := FALSE, PT := #NoDelayTime);
   "Unit1.Em7.Alarms".productionWarning[0] := "Unit1.Em7.Alarms".tonProductionWarning[0].Q;
END_REGION

REGION Network 90: PFE Tooling Warnings 0
   RUNG wire#powerrail
      Contact( FALSE )
      { S7_Templates := "time_type := Time" } "Unit1.Em7.Alarms".tonToolingWarning[0].TON(pt := #NoDelayTime, et =>)
      Coil( "Unit1.Em7.Alarms".toolingWarning[0] )
   END_RUNG
   // the same network as SCL:
   "Unit1.Em7.Alarms".tonToolingWarning[0].TON(IN := FALSE, PT := #NoDelayTime);
   "Unit1.Em7.Alarms".toolingWarning[0] := "Unit1.Em7.Alarms".tonToolingWarning[0].Q;
END_REGION

REGION Network 91: *************** Status ***************************
END_REGION

REGION Network 92: PFE Maintenance Status 0
   RUNG wire#powerrail
      Contact( FALSE )
      Coil( "Unit1.Em7.Alarms".maintenanceStatus[0] )
   END_RUNG
   // the same network as SCL:
   "Unit1.Em7.Alarms".maintenanceStatus[0] := FALSE;
END_REGION

REGION Network 93: PFE Maintenance Status 1
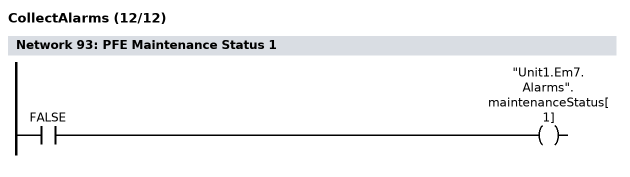
   RUNG wire#powerrail
      Contact( FALSE )
      Coil( "Unit1.Em7.Alarms".maintenanceStatus[1] )
   END_RUNG
   // the same network as SCL:
   "Unit1.Em7.Alarms".maintenanceStatus[1] := FALSE;
END_REGION
END_FUNCTION
